GLOBALCONSTANTS Computers (* Global constants *)
  (* Standard: 61499-1; Description: Copyright (c) 2023 HR Agrartechnik GmbH This program and the accompanying materials are made available under the terms of the Eclipse Public License 2.0 which is available at https://www.eclipse.org/legal/epl-2.0/ SPDX-License-Identifier: EPL-2.0 *)
  (* Version 1.0, 2023-10-22, Franz Höpfinger, HR Agrartechnik GmbH *)
  PACKAGE stations;
  VAR_GLOBAL CONSTANT
    C_LO : WSTRING := "localhost:61499";
    C_ET : WSTRING := "192.168.5.1:61499";
    C_ST : WSTRING := "192.168.4.1:61499";
    C_00 : WSTRING := "192.168.4.1:61499";
  END_VAR
END_GLOBALCONSTANTS
